{attribute 'qualified_only'}
VAR_GLOBAL
	bEnableSimulation : BOOL;
	bStartSimulation : BOOL;
	bAutoMode : BOOL;
	fManualCylinderPositionReference : REAL;
	fCylinderVelocityReference : REAL;
END_VAR

(* stored: Version 1.1.0.1, ProductVersion 3.1.4024.10
   GVL Inputs: Id {e951088c-709d-404f-bb3e-4c135570158d} *)
